// TIA Portal V16 export
// export: Created 2024-09-05T15:58:41.4102112Z, ExportSetting WithDefaults, DisplayName Totally Integrated Automation Portal, DisplayVersion V16 Update 6, DisplayName TIA Portal Version Control Interface, DisplayVersion V16 Update 2, DisplayName TIA Portal Openness, DisplayVersion V16 Update 6, DisplayName STEP 7 Professional, DisplayVersion V16 Update 6, DisplayName STEP 7 Safety, DisplayVersion V16, DisplayName WinCC Advanced, DisplayVersion V16 Update 6
VAR_GLOBAL   // PLC tag table "Default tag table"
   tAirPressureOK AT %T0 : Timer;
   INIT_SCAN AT %M2.0 : Bool;
   ALARMA_0 AT %MW4 : Int;
   ALARMA_1 AT %MW6 : Int;
   ALARMA_2 AT %MW8 : Int;
   ALARMA_3 AT %MW10 : Int;
   ALARMA_4 AT %MW12 : Int;
   ALARMA_5 AT %MW14 : Int;
   "ALARMA ACTIVA" AT %M2.1 : Bool;
   ALARM_AKCNOWLEDGE AT %M2.2 : Bool;
   SENSOR_LASER_DER AT %I11.4 : Bool;
   SENSOR_LASER_IZQ AT %I11.5 : Bool;
END_VAR
VAR_GLOBAL CONSTANT   // user constants
   NumberOfEksKeys : Int := 100;
   NumberOfEksEngineerKeys : Int := 5;
   GapLeaderLevel : Int := 2;
   MaintenanceLevel : Int := 3;
   EngineerLevel : Int := 5;
   NumberOfProductionPrograms : UInt := 8;
   NumberOfProductionProducts : Int := 8;
   LoggerBufferSize : Int := 32;
   LoggerTypeAlarm : Int := 1;
   LoggerTypeStatus : Int := 2;
   LoggerNumberOfPartErrors : Int := 5;
   LoggerTypePart : Int := 3;
   LoggerTypeUser : Int := 4;
   LoggerTypeComment : Int := 99;
   AlarmsCount : Int := 256;
   NumberOfIJCoreMessages : Int := 30;
   LoggerTypeRiveting : Int := 50;
   EksNumberOfKeys : Int := 100;
   EksNumberOfEngineerKeys : Int := 50;
   EksGapLeaderLevel : Int := 2;
   EksMaintenanceLevel : Int := 3;
   EksEngineerLevel : Int := 5;
END_VAR
